FUNCTION_BLOCK FB_AGGREGATION
VAR_INPUT
	//fbImplication: REFERENCE TO FB_IMPLICATION;
	Myrules:ARRAY [1..NumOfFisRules] OF FIS_RULES;
	MyFISoutputs:ARRAY [1..NumOfFISOutputs] OF FIS_VAR;
	X:REAL;
END_VAR

VAR
	firstRule,LastRule,i,j:DINT;
	aofFuzzySet:  ARRAY [1..NumOfFisRules] OF REAL;
	fbImplication:FB_IMPLICATION;
	MyMF: INT;
END_VAR
VAR_OUTPUT
	FSValue:REAL; 
END_VAR

//firstRule:=LOWER_BOUND(Rule,1);
//LastRule:=UPPER_BOUND(Rule,1);
//FOR i:=firstRule TO LastRule DO
FOR i:=1 TO NumOfFisRules DO
	FOR j:=1 TO NumOfFISOutputs DO
		IF Myrules[i].Consequents[j]>0 THEN
		MyMF:=Myrules[i].Consequents[j];
		fbImplication(
				X:=X,
				Antecedent:=Myrules[i].Antecedent,
				FISOutputMf:= MyFISoutputs[j].MF[MyMF]);
		aofFuzzySet[i]:=fbImplication.RuleFuzzySet;
		END_IF
	END_FOR
END_FOR

FSValue:=FuzzyOR_array(maximum,aofFuzzySet);

END_FUNCTION_BLOCK

(* stored: Version 1.1.0.1, ProductVersion 3.1.4024.6
   POU FB_AGGREGATION: Id {82675cbe-95f4-4a61-93e4-f185b93b6fec}, SpecialFunc None *)
